# EPICS autosave request: IOCs/MS_DAQ/MSApp/Db/MS_Support_settings.req
# This file is used by autosave to determine what PVs to save (currently, autosave not used)
# It is also used by MS DAQ to determine what PVs to create

# This file contains all of the PVs used by the MS.

####################
# Time PVs
####################

$(P)$(R)CreationTimeSupportName
$(P)$(R)ProgIntSupportName
